INTERFACE I_Testsuites EXTENDS I_Base

PROPERTY PUBLIC P_Data : reference to ST_Testsuites
GET
END_GET
END_PROPERTY

PROPERTY PUBLIC P_List : I_ListSTRING
GET
END_GET
END_PROPERTY

PROPERTY PUBLIC P_Options : REFERENCE TO ST_TestsuitesOptions
GET
END_GET
END_PROPERTY

END_INTERFACE

(* stored: Version 1.1.0.1
   Itf I_Testsuites: Id {606cd2f2-cac2-4517-8699-c23aaa0c4b09}
   Property P_Data: Id {85c32222-d556-0312-20e5-4473baafbb98}
   Get Get: Id {50c617ac-7957-0d8c-29c1-501d545160bb}
   Property P_List: Id {2894c1aa-7a7c-0cc9-216c-5c628c5f3c09}
   Get Get: Id {cf580b2f-d72c-0b8a-01bc-4c4ee7bcbb85}
   Property P_Options: Id {cac67df2-87b6-04eb-1648-4410cde413cc}
   Get Get: Id {9f9c64ea-3b7f-00ce-05a0-5c3ad432879f} *)
